RESOURCE_TYPE _WaterHeaterPlant
  (* Standard: 61499-2 *)
  (* Version 0.1, 2017-00-25, hpea485, UOA *)
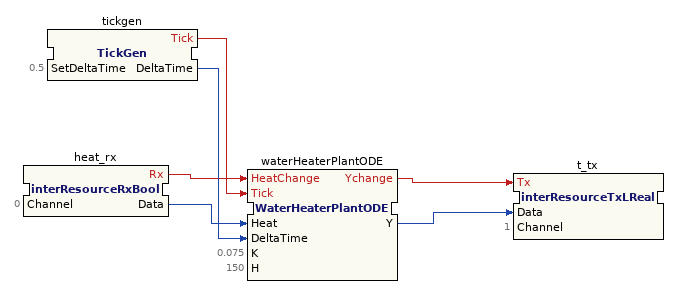
  FBS
    waterHeaterPlantODE : WaterHeaterPlantODE(K := 0.075, H := 150);
    t_tx : interResourceTxLReal(Channel := 1);
    heat_rx : interResourceRxBool(Channel := 0);
    tickgen : TickGen(SetDeltaTime := 0.5);
  END_FBS
  EVENT_CONNECTIONS
    waterHeaterPlantODE.Ychange TO t_tx.Tx;
    heat_rx.Rx TO waterHeaterPlantODE.HeatChange;
    tickgen.Tick TO waterHeaterPlantODE.Tick;
  END_CONNECTIONS
  DATA_CONNECTIONS
    waterHeaterPlantODE.Y TO t_tx.Data;
    heat_rx.Data TO waterHeaterPlantODE.Heat;
    tickgen.DeltaTime TO waterHeaterPlantODE.DeltaTime;
  END_CONNECTIONS
END_RESOURCE_TYPE
